// TIA Portal V17 export
// export: Created 2023-12-22T15:05:25.4356009Z, ExportSetting WithDefaults, DisplayName Totally Integrated Automation Portal, DisplayVersion V17, DisplayName TIA Portal Openness, DisplayVersion V17, DisplayName TIA Portal Version Control Interface, DisplayVersion V17, DisplayName STEP 7 Professional, DisplayVersion V17, DisplayName STEP 7 Safety, DisplayVersion V17, DisplayName WinCC Advanced, DisplayVersion V17
FUNCTION_BLOCK "Logick"   // FB1, LAD
{ S7_Optimized_Access := 'FALSE' }
VERSION : 0.1
// stored: AutoNumber true, IsIECCheckEnabled false, SetENOAutomatically false, UDAEnableTagReadback false
   VAR DB_SPECIFIC
      Start_ELZ : Bool;   // Запуск электролизеров (приготовления)
      REQ_Wash : Bool;   // Запрос запуска промывки
      Force_Wash : Bool;   // Принудительная промывка
      ELZ : Bool;
      Local : Bool;   // Дистанционное управление
      Step_Wash : Int;   // Шаг промывки
      ELZ_LED : Int;   // Подсветка электролизера на панели
      RM_1 { S7_SetPoint := 'True'} : Real;
      Alarm : Word;   // Слово аварий
      Alarms : Struct
         Gas : Bool;   // Остановка по загазованности
         ELZ_AHLS : Bool;   // Электролизер - переполнение поддона
      END_STRUCT;
   END_VAR
   VAR
      ELZ_1 { S7_SetPoint := 'True'} : "ELZ";
   END_VAR
   VAR DB_SPECIFIC
      Days : Struct   // Расписание промывки (дни)
         D_1 : Bool;   // Расписание промывки (день 1)
         D_2 : Bool;   // Расписание промывки (день 2)
         D_3 : Bool;   // Расписание промывки (день 3)
         D_4 : Bool;   // Расписание промывки (день 4)
         D_5 : Bool;   // Расписание промывки (день 5)
         D_6 : Bool;   // Расписание промывки (день 6)
         D_7 : Bool;   // Расписание промывки (день 7)
      END_STRUCT;
      Houres : Struct   // Расписание промывки (часы)
         H_D_1 : Int;   // Расписание промывки (часы 1 дня)
         H_D_2 : Int;   // Расписание промывки (часы 2 дня)
         H_D_3 : Int;   // Расписание промывки (часы 3 дня)
         H_D_4 : Int;   // Расписание промывки (часы 4 дня)
         H_D_5 : Int;   // Расписание промывки (часы 5 дня)
         H_D_6 : Int;   // Расписание промывки (часы 6 дня)
         H_D_7 : Int;   // Расписание промывки (часы 7 дня)
      END_STRUCT;
      Minutes : Struct   // Расписание промывки (минуты)
         M_D_1 : Int;   // Расписание промывки (минуты 1 дня)
         M_D_2 : Int;   // Расписание промывки (минуты 2 дня)
         M_D_3 : Int;   // Расписание промывки (минуты 3 дня)
         M_D_4 : Int;   // Расписание промывки (минуты 4 дня)
         M_D_5 : Int;   // Расписание промывки (минуты 5 дня)
         M_D_6 : Int;   // Расписание промывки (минуты 6 дня)
         M_D_7 : Int;   // Расписание промывки (минуты 7 дня)
      END_STRUCT;
   END_VAR
   VAR
      T_Wash { S7_SetPoint := 'True'} : "Time_M";   // Время промывки
   END_VAR
   VAR_TEMP   // added for the SCL form of the ladder/FBD networks
      _w1 : Bool;
      _w2 : Bool;
   END_VAR
BEGIN

REGION Network 1: Электролизеры
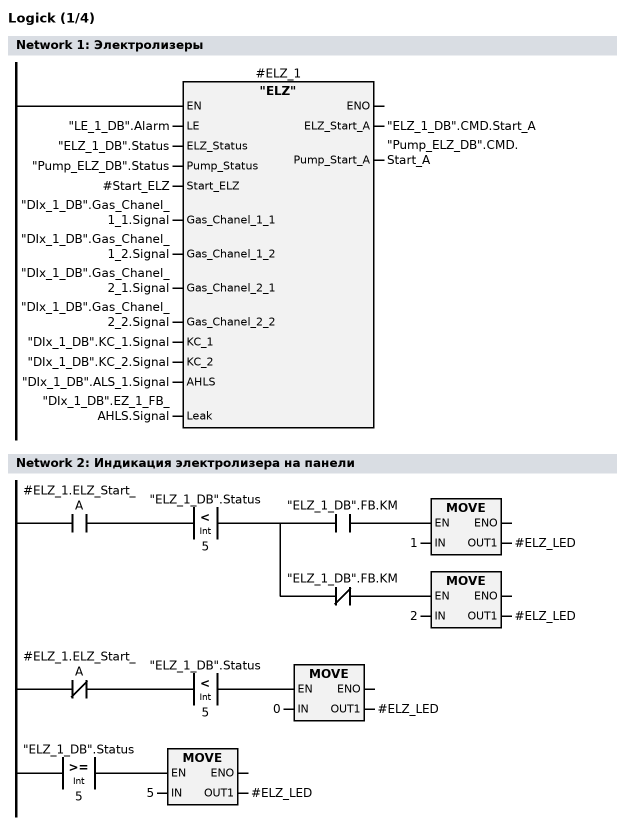
   RUNG wire#powerrail
      #ELZ_1(LE := "LE_1_DB".Alarm, ELZ_Status := "ELZ_1_DB".Status, Pump_Status := "Pump_ELZ_DB".Status, Start_ELZ := #Start_ELZ, Gas_Chanel_1_1 := "DIx_1_DB".Gas_Chanel_1_1.Signal, Gas_Chanel_1_2 := "DIx_1_DB".Gas_Chanel_1_2.Signal, Gas_Chanel_2_1 := "DIx_1_DB".Gas_Chanel_2_1.Signal, Gas_Chanel_2_2 := "DIx_1_DB".Gas_Chanel_2_2.Signal, KC_1 := "DIx_1_DB".KC_1.Signal, KC_2 := "DIx_1_DB".KC_2.Signal, AHLS := "DIx_1_DB".ALS_1.Signal, Leak := "DIx_1_DB".EZ_1_FB_AHLS.Signal, ELZ_Start_A => "ELZ_1_DB".CMD.Start_A, Pump_Start_A => "Pump_ELZ_DB".CMD.Start_A)
   END_RUNG
   // the same network as SCL:
   #ELZ_1(LE := "LE_1_DB".Alarm,   // "ELZ"
          ELZ_Status := "ELZ_1_DB".Status,
          Pump_Status := "Pump_ELZ_DB".Status,
          Start_ELZ := #Start_ELZ,
          Gas_Chanel_1_1 := "DIx_1_DB".Gas_Chanel_1_1.Signal,
          Gas_Chanel_1_2 := "DIx_1_DB".Gas_Chanel_1_2.Signal,
          Gas_Chanel_2_1 := "DIx_1_DB".Gas_Chanel_2_1.Signal,
          Gas_Chanel_2_2 := "DIx_1_DB".Gas_Chanel_2_2.Signal,
          KC_1 := "DIx_1_DB".KC_1.Signal,
          KC_2 := "DIx_1_DB".KC_2.Signal,
          AHLS := "DIx_1_DB".ALS_1.Signal,
          Leak := "DIx_1_DB".EZ_1_FB_AHLS.Signal,
          ELZ_Start_A => "ELZ_1_DB".CMD.Start_A,
          Pump_Start_A => "Pump_ELZ_DB".CMD.Start_A);
END_REGION

REGION Network 2: Индикация электролизера на панели
   RUNG wire#powerrail
      Contact( #ELZ_1.ELZ_Start_A )
      { S7_Templates := "SrcType := Int" } LT_Contact(in1 := "ELZ_1_DB".Status, in2 := 5)
      wire#w1
      Contact( "ELZ_1_DB".FB.KM )
      Move(in := 1, out1 => #ELZ_LED)
   END_RUNG
   RUNG wire#w1
      I_Contact( "ELZ_1_DB".FB.KM )
      Move(in := 2, out1 => #ELZ_LED)
   END_RUNG
   RUNG wire#powerrail
      I_Contact( #ELZ_1.ELZ_Start_A )
      { S7_Templates := "SrcType := Int" } LT_Contact(in1 := "ELZ_1_DB".Status, in2 := 5)
      Move(in := 0, out1 => #ELZ_LED)
   END_RUNG
   RUNG wire#powerrail
      { S7_Templates := "SrcType := Int" } GE_Contact(in1 := "ELZ_1_DB".Status, in2 := 5)
      Move(in := 5, out1 => #ELZ_LED)
   END_RUNG
   // the same network as SCL:
   #_w1 := #ELZ_1.ELZ_Start_A AND ("ELZ_1_DB".Status < 5);
   IF #_w1 AND "ELZ_1_DB".FB.KM THEN #ELZ_LED := 1; END_IF;
   IF #_w1 AND NOT "ELZ_1_DB".FB.KM THEN #ELZ_LED := 2; END_IF;
   IF NOT #ELZ_1.ELZ_Start_A AND ("ELZ_1_DB".Status < 5) THEN #ELZ_LED := 0; END_IF;
   IF "ELZ_1_DB".Status >= 5 THEN #ELZ_LED := 5; END_IF;
END_REGION

REGION Network 3: Запрос промывки фильтров (Пришло время в расписании)
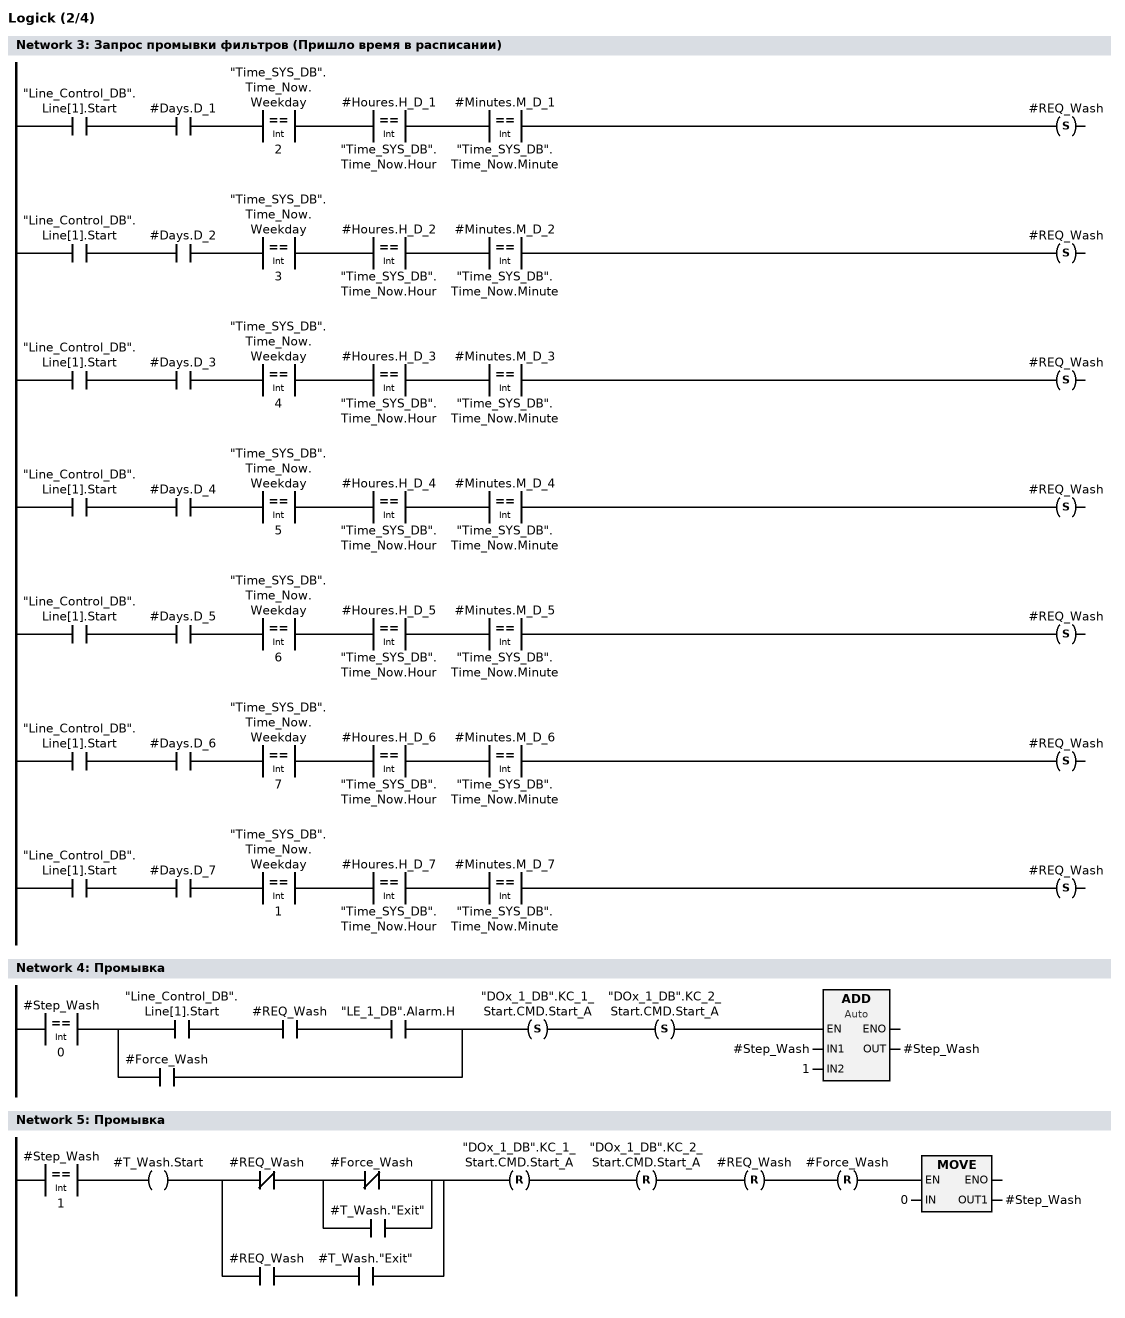
   RUNG wire#powerrail
      Contact( "Line_Control_DB".Line[1].Start )
      Contact( #Days.D_1 )
      { S7_Templates := "SrcType := Int" } EQ_Contact(in1 := "Time_SYS_DB".Time_Now.Weekday, in2 := 2)
      { S7_Templates := "SrcType := Int" } EQ_Contact(in1 := #Houres.H_D_1, in2 := "Time_SYS_DB".Time_Now.Hour)
      { S7_Templates := "SrcType := Int" } EQ_Contact(in1 := #Minutes.M_D_1, in2 := "Time_SYS_DB".Time_Now.Minute)
      S_Coil( #REQ_Wash )
   END_RUNG
   RUNG wire#powerrail
      Contact( "Line_Control_DB".Line[1].Start )
      Contact( #Days.D_2 )
      { S7_Templates := "SrcType := Int" } EQ_Contact(in1 := "Time_SYS_DB".Time_Now.Weekday, in2 := 3)
      { S7_Templates := "SrcType := Int" } EQ_Contact(in1 := #Houres.H_D_2, in2 := "Time_SYS_DB".Time_Now.Hour)
      { S7_Templates := "SrcType := Int" } EQ_Contact(in1 := #Minutes.M_D_2, in2 := "Time_SYS_DB".Time_Now.Minute)
      S_Coil( #REQ_Wash )
   END_RUNG
   RUNG wire#powerrail
      Contact( "Line_Control_DB".Line[1].Start )
      Contact( #Days.D_3 )
      { S7_Templates := "SrcType := Int" } EQ_Contact(in1 := "Time_SYS_DB".Time_Now.Weekday, in2 := 4)
      { S7_Templates := "SrcType := Int" } EQ_Contact(in1 := #Houres.H_D_3, in2 := "Time_SYS_DB".Time_Now.Hour)
      { S7_Templates := "SrcType := Int" } EQ_Contact(in1 := #Minutes.M_D_3, in2 := "Time_SYS_DB".Time_Now.Minute)
      S_Coil( #REQ_Wash )
   END_RUNG
   RUNG wire#powerrail
      Contact( "Line_Control_DB".Line[1].Start )
      Contact( #Days.D_4 )
      { S7_Templates := "SrcType := Int" } EQ_Contact(in1 := "Time_SYS_DB".Time_Now.Weekday, in2 := 5)
      { S7_Templates := "SrcType := Int" } EQ_Contact(in1 := #Houres.H_D_4, in2 := "Time_SYS_DB".Time_Now.Hour)
      { S7_Templates := "SrcType := Int" } EQ_Contact(in1 := #Minutes.M_D_4, in2 := "Time_SYS_DB".Time_Now.Minute)
      S_Coil( #REQ_Wash )
   END_RUNG
   RUNG wire#powerrail
      Contact( "Line_Control_DB".Line[1].Start )
      Contact( #Days.D_5 )
      { S7_Templates := "SrcType := Int" } EQ_Contact(in1 := "Time_SYS_DB".Time_Now.Weekday, in2 := 6)
      { S7_Templates := "SrcType := Int" } EQ_Contact(in1 := #Houres.H_D_5, in2 := "Time_SYS_DB".Time_Now.Hour)
      { S7_Templates := "SrcType := Int" } EQ_Contact(in1 := #Minutes.M_D_5, in2 := "Time_SYS_DB".Time_Now.Minute)
      S_Coil( #REQ_Wash )
   END_RUNG
   RUNG wire#powerrail
      Contact( "Line_Control_DB".Line[1].Start )
      Contact( #Days.D_6 )
      { S7_Templates := "SrcType := Int" } EQ_Contact(in1 := "Time_SYS_DB".Time_Now.Weekday, in2 := 7)
      { S7_Templates := "SrcType := Int" } EQ_Contact(in1 := #Houres.H_D_6, in2 := "Time_SYS_DB".Time_Now.Hour)
      { S7_Templates := "SrcType := Int" } EQ_Contact(in1 := #Minutes.M_D_6, in2 := "Time_SYS_DB".Time_Now.Minute)
      S_Coil( #REQ_Wash )
   END_RUNG
   RUNG wire#powerrail
      Contact( "Line_Control_DB".Line[1].Start )
      Contact( #Days.D_7 )
      { S7_Templates := "SrcType := Int" } EQ_Contact(in1 := "Time_SYS_DB".Time_Now.Weekday, in2 := 1)
      { S7_Templates := "SrcType := Int" } EQ_Contact(in1 := #Houres.H_D_7, in2 := "Time_SYS_DB".Time_Now.Hour)
      { S7_Templates := "SrcType := Int" } EQ_Contact(in1 := #Minutes.M_D_7, in2 := "Time_SYS_DB".Time_Now.Minute)
      S_Coil( #REQ_Wash )
   END_RUNG
   // the same network as SCL:
   IF "Line_Control_DB".Line[1].Start AND #Days.D_1 AND ("Time_SYS_DB".Time_Now.Weekday = 2) AND (#Houres.H_D_1 = "Time_SYS_DB".Time_Now.Hour) AND (#Minutes.M_D_1 = "Time_SYS_DB".Time_Now.Minute) THEN
       #REQ_Wash := TRUE;
   END_IF;
   IF "Line_Control_DB".Line[1].Start AND #Days.D_2 AND ("Time_SYS_DB".Time_Now.Weekday = 3) AND (#Houres.H_D_2 = "Time_SYS_DB".Time_Now.Hour) AND (#Minutes.M_D_2 = "Time_SYS_DB".Time_Now.Minute) THEN
       #REQ_Wash := TRUE;
   END_IF;
   IF "Line_Control_DB".Line[1].Start AND #Days.D_3 AND ("Time_SYS_DB".Time_Now.Weekday = 4) AND (#Houres.H_D_3 = "Time_SYS_DB".Time_Now.Hour) AND (#Minutes.M_D_3 = "Time_SYS_DB".Time_Now.Minute) THEN
       #REQ_Wash := TRUE;
   END_IF;
   IF "Line_Control_DB".Line[1].Start AND #Days.D_4 AND ("Time_SYS_DB".Time_Now.Weekday = 5) AND (#Houres.H_D_4 = "Time_SYS_DB".Time_Now.Hour) AND (#Minutes.M_D_4 = "Time_SYS_DB".Time_Now.Minute) THEN
       #REQ_Wash := TRUE;
   END_IF;
   IF "Line_Control_DB".Line[1].Start AND #Days.D_5 AND ("Time_SYS_DB".Time_Now.Weekday = 6) AND (#Houres.H_D_5 = "Time_SYS_DB".Time_Now.Hour) AND (#Minutes.M_D_5 = "Time_SYS_DB".Time_Now.Minute) THEN
       #REQ_Wash := TRUE;
   END_IF;
   IF "Line_Control_DB".Line[1].Start AND #Days.D_6 AND ("Time_SYS_DB".Time_Now.Weekday = 7) AND (#Houres.H_D_6 = "Time_SYS_DB".Time_Now.Hour) AND (#Minutes.M_D_6 = "Time_SYS_DB".Time_Now.Minute) THEN
       #REQ_Wash := TRUE;
   END_IF;
   IF "Line_Control_DB".Line[1].Start AND #Days.D_7 AND ("Time_SYS_DB".Time_Now.Weekday = 1) AND (#Houres.H_D_7 = "Time_SYS_DB".Time_Now.Hour) AND (#Minutes.M_D_7 = "Time_SYS_DB".Time_Now.Minute) THEN
       #REQ_Wash := TRUE;
   END_IF;
END_REGION

REGION Network 4: Промывка
   RUNG wire#powerrail
      { S7_Templates := "SrcType := Int" } EQ_Contact(in1 := #Step_Wash, in2 := 0)
      wire#w1
      Contact( "Line_Control_DB".Line[1].Start )
      Contact( #REQ_Wash )
      Contact( "LE_1_DB".Alarm.H )
      wire#w2
      S_Coil( "DOx_1_DB".KC_1_Start.CMD.Start_A )
      S_Coil( "DOx_1_DB".KC_2_Start.CMD.Start_A )
      Add(in1 := #Step_Wash, in2 := 1, out => #Step_Wash)
   END_RUNG
   RUNG wire#w1
      Contact( #Force_Wash )
   END_RUNG wire#w2
   // the same network as SCL:
   IF (#Step_Wash = 0) AND (("Line_Control_DB".Line[1].Start AND #REQ_Wash AND "LE_1_DB".Alarm.H) OR #Force_Wash) THEN
       "DOx_1_DB".KC_1_Start.CMD.Start_A := TRUE;
       "DOx_1_DB".KC_2_Start.CMD.Start_A := TRUE;
       #Step_Wash := #Step_Wash + 1;
   END_IF;
END_REGION

REGION Network 5: Промывка
   RUNG wire#powerrail
      { S7_Templates := "SrcType := Int" } EQ_Contact(in1 := #Step_Wash, in2 := 1)
      Coil( #T_Wash.Start )
      wire#w1
      I_Contact( #REQ_Wash )
      wire#w2
      I_Contact( #Force_Wash )
      wire#w3
      R_Coil( "DOx_1_DB".KC_1_Start.CMD.Start_A )
      R_Coil( "DOx_1_DB".KC_2_Start.CMD.Start_A )
      R_Coil( #REQ_Wash )
      R_Coil( #Force_Wash )
      Move(in := 0, out1 => #Step_Wash)
   END_RUNG
   RUNG wire#w2
      Contact( #T_Wash."Exit" )
   END_RUNG wire#w3
   RUNG wire#w1
      Contact( #REQ_Wash )
      Contact( #T_Wash."Exit" )
   END_RUNG wire#w3
   // the same network as SCL:
   #T_Wash.Start := #Step_Wash = 1;
   IF #T_Wash.Start AND ((NOT #REQ_Wash AND (NOT #Force_Wash OR #T_Wash."Exit")) OR (#REQ_Wash AND #T_Wash."Exit")) THEN
       "DOx_1_DB".KC_1_Start.CMD.Start_A := FALSE;
       "DOx_1_DB".KC_2_Start.CMD.Start_A := FALSE;
   END_IF;
   #_w1 := #T_Wash.Start AND ((NOT #REQ_Wash AND (NOT #Force_Wash OR #T_Wash."Exit")) OR (#REQ_Wash AND #T_Wash."Exit"));
   IF #_w1 THEN
       #REQ_Wash := FALSE;
       #Force_Wash := FALSE;
       #Step_Wash := 0;
   END_IF;
END_REGION

REGION Network 6: Блокировка и авария насосов 1 и 2 по низкому уровню и неисправности датчиков
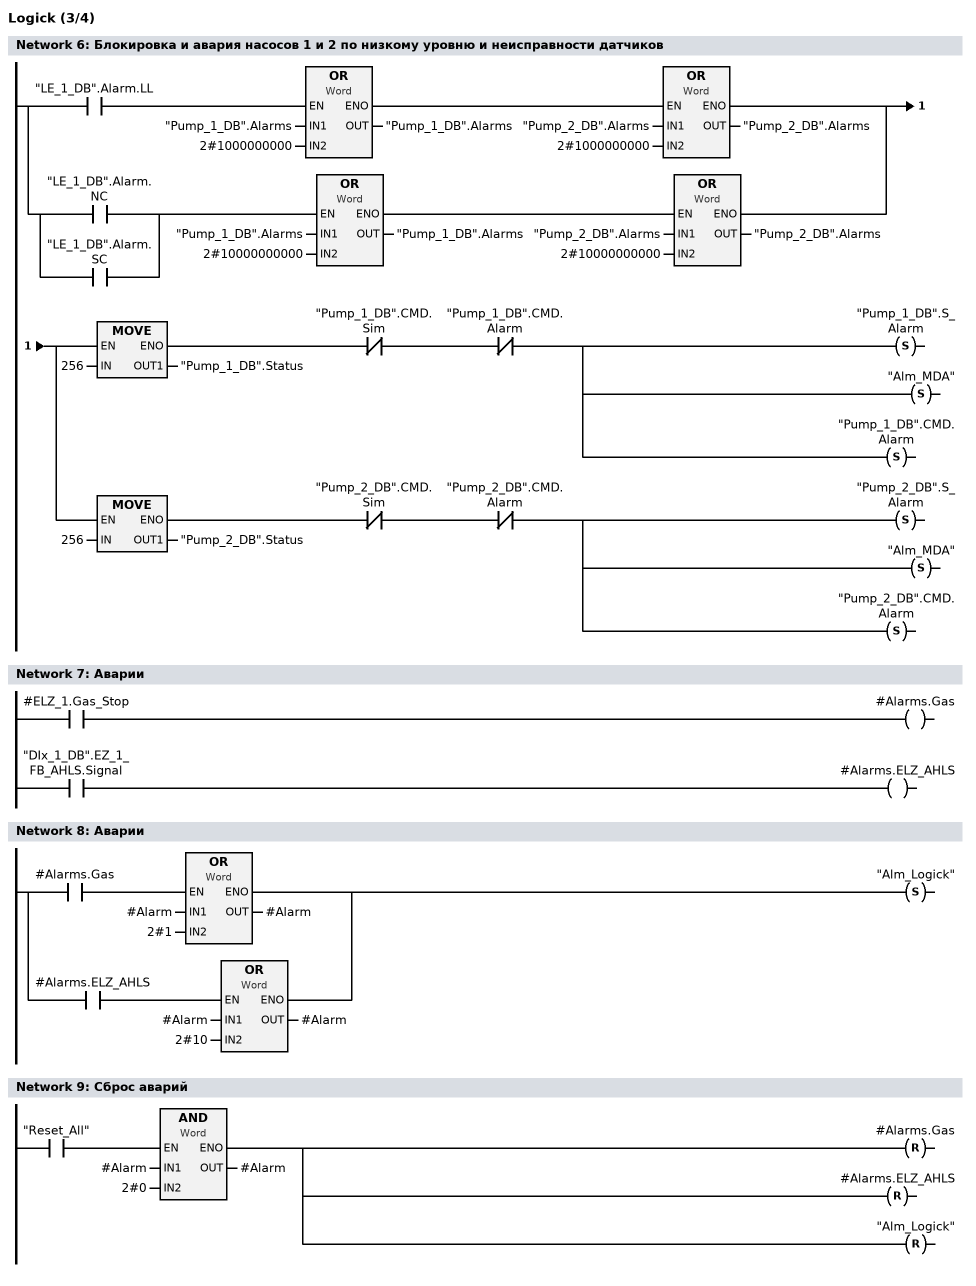
   // ENO of a box is taken as its EN; it also drops when the box reports an error
   IF "LE_1_DB".Alarm.LL THEN
       "Pump_1_DB".Alarms := "Pump_1_DB".Alarms OR 2#1000000000;
       "Pump_2_DB".Alarms := "Pump_2_DB".Alarms OR 2#1000000000;
   END_IF;
   #_w1 := "LE_1_DB".Alarm.NC OR "LE_1_DB".Alarm.SC;
   IF #_w1 THEN
       "Pump_1_DB".Alarms := "Pump_1_DB".Alarms OR 2#10000000000;
       "Pump_2_DB".Alarms := "Pump_2_DB".Alarms OR 2#10000000000;
   END_IF;
   #_w2 := "LE_1_DB".Alarm.LL OR #_w1;
   IF #_w2 THEN "Pump_1_DB".Status := 256; END_IF;
   IF #_w2 AND NOT "Pump_1_DB".CMD.Sim AND NOT "Pump_1_DB".CMD.Alarm THEN
       "Pump_1_DB".S_Alarm := TRUE;
       "Alm_MDA" := TRUE;
       "Pump_1_DB".CMD.Alarm := TRUE;
   END_IF;
   IF #_w2 THEN "Pump_2_DB".Status := 256; END_IF;
   IF #_w2 AND NOT "Pump_2_DB".CMD.Sim AND NOT "Pump_2_DB".CMD.Alarm THEN
       "Pump_2_DB".S_Alarm := TRUE;
       "Alm_MDA" := TRUE;
       "Pump_2_DB".CMD.Alarm := TRUE;
   END_IF;
END_REGION

REGION Network 7: Аварии
   RUNG wire#powerrail
      Contact( #ELZ_1.Gas_Stop )
      Coil( #Alarms.Gas )
   END_RUNG
   RUNG wire#powerrail
      Contact( "DIx_1_DB".EZ_1_FB_AHLS.Signal )
      Coil( #Alarms.ELZ_AHLS )
   END_RUNG
   // the same network as SCL:
   #Alarms.Gas := #ELZ_1.Gas_Stop;
   #Alarms.ELZ_AHLS := "DIx_1_DB".EZ_1_FB_AHLS.Signal;
END_REGION

REGION Network 8: Аварии
   IF #Alarms.Gas THEN #Alarm := #Alarm OR 2#1; END_IF;
   IF #Alarms.ELZ_AHLS THEN #Alarm := #Alarm OR 2#10; END_IF;
   IF #Alarms.Gas OR #Alarms.ELZ_AHLS THEN "Alm_Logick" := TRUE; END_IF;
END_REGION

REGION Network 9: Сброс аварий
   RUNG wire#powerrail
      Contact( "Reset_All" )
      { S7_Templates := "SrcType := Word"; S7_GenerateENO := "TRUE" } And(in1 := #Alarm, in2 := 2#0, out => #Alarm)
      wire#w1
      R_Coil( #Alarms.Gas )
   END_RUNG
   RUNG wire#w1
      R_Coil( #Alarms.ELZ_AHLS )
   END_RUNG
   RUNG wire#w1
      R_Coil( "Alm_Logick" )
   END_RUNG
   // the same network as SCL:
   IF "Reset_All" THEN
       #Alarm := #Alarm AND 2#0;
       #Alarms.Gas := FALSE;
       #Alarms.ELZ_AHLS := FALSE;
       "Alm_Logick" := FALSE;
   END_IF;
END_REGION

REGION Network 10: Сигнальная колонна
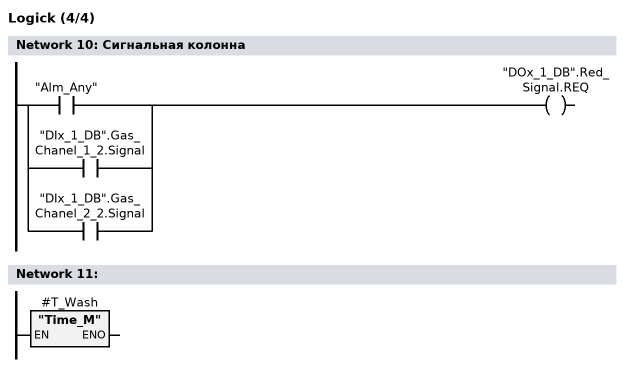
   RUNG wire#powerrail
      Contact( "Alm_Any" )
      wire#w1
      Coil( "DOx_1_DB".Red_Signal.REQ )
   END_RUNG
   RUNG wire#powerrail
      Contact( "DIx_1_DB".Gas_Chanel_1_2.Signal )
   END_RUNG wire#w1
   RUNG wire#powerrail
      Contact( "DIx_1_DB".Gas_Chanel_2_2.Signal )
   END_RUNG wire#w1
   // the same network as SCL:
   "DOx_1_DB".Red_Signal.REQ := "Alm_Any" OR "DIx_1_DB".Gas_Chanel_1_2.Signal OR "DIx_1_DB".Gas_Chanel_2_2.Signal;
END_REGION

REGION Network 11
   RUNG wire#powerrail
      #T_Wash()
   END_RUNG
   // the same network as SCL:
   #T_Wash();   // "Time_M"
END_REGION
END_FUNCTION_BLOCK
